FUNCTION_BLOCK TrackingLogic
VAR_INPUT
END_VAR
VAR_OUTPUT
END_VAR
VAR
END_VAR



IF GVL.Position[0].Occupied  THEN
	IF GVL.Position[0].Done THEN
		GVL.Position[0].Done := FALSE;
		GVL.Position[1].Piece := GVL.Position[0].Piece;
		GVL.Position[1].Occupied := TRUE;
		GVL.Position[0].Occupied := FALSE;
		GVL.Position[1].Done := FALSE;
	END_IF
END_IF

IF GVL.Position[1].Occupied  THEN
	IF GVL.Position[1].Done THEN
		GVL.Position[1].Done := FALSE;
		GVL.Position[2].Piece := GVL.Position[1].Piece;
		GVL.Position[2].Occupied := TRUE;
		GVL.Position[1].Occupied := FALSE;
		GVL.Position[2].Done := FALSE;
		GVL.Position[2].Processed := FALSE;
	END_IF
END_IF

IF GVL.Position[2].Occupied  THEN
	IF GVL.Position[2].Done THEN
		//GVL.Position[2].Processed := FALSE;
		GVL.Position[3].Done := FALSE;
		GVL.Position[2].Occupied := FALSE;
		GVL.Position[3].Piece := GVL.Position[2].Piece;
		GVL.Position[3].Occupied := TRUE;
		GVL.Position[2].Done := FALSE;
	END_IF
END_IF

IF GVL.Position[3].Occupied  THEN
	IF GVL.Position[3].Done THEN
		GVL.Position[3].Done := FALSE;
		GVL.Position[4].Piece := GVL.Position[3].Piece;
		GVL.Position[4].Occupied := TRUE;
		GVL.Position[3].Occupied := FALSE;
		GVL.Position[4].Done := FALSE;
	END_IF
END_IF

IF GVL.Position[4].Occupied  THEN
	IF GVL.Position[4].Done THEN
		GVL.Position[4].Done := FALSE;
		GVL.Position[5].Piece := GVL.Position[4].Piece;
		GVL.Position[5].Occupied := TRUE;
		GVL.Position[4].Occupied := FALSE;
		GVL.Position[5].Done := FALSE;
	END_IF
END_IF

IF GVL.Position[5].Occupied  THEN
	IF GVL.Position[5].Done THEN
		GVL.Position[5].Done := FALSE;
		GVL.Position[5].Occupied := FALSE;
	END_IF
END_IF

END_FUNCTION_BLOCK

(* stored: Version 1.1.0.1, ProductVersion 3.1.4024.12
   POU TrackingLogic: Id {e099012d-54a4-4c6c-bcf9-8781338d3583}, SpecialFunc None *)
